TYPE ST_LA_Steuerung :
STRUCT
	Anforderung_Lueftung_Halle 							: BOOL := FALSE; (*manuell gesetzt*)
	Anforderung_Lueftung_Seminarraum					: BOOL := FALSE; (*manuell gesetzt*)
	Anforderung_Lueftung_Halle_ueber_Nutzungszeit 		: BOOL := FALSE; (*manuell gesetzt*)
	Anforderung_Lueftung_Seminarraum_ueber_CO2_Grenzwert: BOOL := TRUE; (*manuell gesetzt*)
	Anforderung_Lueftung_Seminarraum_ueber_Nutzungszeit : BOOL := FALSE; (*manuell gesetzt*)
	Entriegelung_Anlage 								: BOOL := FALSE; (*manuell gesetzt*)
	Sollwertauswahl_Anlage 								: BOOL := FALSE; (*manuell gesetzt*)
END_STRUCT
END_TYPE

(* stored: Version 1.1.0.1, ProductVersion 3.1.4024.9
   DUT ST_LA_Steuerung: Id {fb10cd66-fb7d-4075-bb42-697d1f76c832} *)
